Staubli VAL3: setConvSpeed.pgx

program setConvSpeed(num x_nConvNum (dimensions=1), num x_nConvSpeed (dimensions=1))
  local num l_nRatio[2]
begin
  // This programs sets, by an analog output, the speed of the
  //  conveyor. The program takes as an input parameter the speed in
  //  mm/s, then it will convert it to the corresponding value that
  //  has to be actually written into the analog output. The local
  //  variable l_nRatio has to be adapted to match the hardware.
  //
  // Input parameters
  //  x_nConvNum      : Conveyor number
  //  x_nConvSpeed    : Conveyor speed in mm/s
  //
  // Output parameters
  //  None            :
  //
  //----------------------------------------------------------------
  //
  l_nRatio[0]=35
  //
  if ioStatus(aConvSpeed[x_nConvNum])>=0
    aioSet(aConvSpeed[x_nConvNum],x_nConvSpeed*l_nRatio[x_nConvNum])
  endIf
  //
end
